// TIA Portal V17 export
// export: Created 2024-09-02T12:50:17.0977902Z, ExportSetting WithDefaults, DisplayName Totally Integrated Automation Portal, DisplayVersion V17, DisplayName TIA Portal Openness, DisplayVersion V17, DisplayName TIA Portal Version Control Interface, DisplayVersion V17, DisplayName STEP 7 Professional, DisplayVersion V17, DisplayName STEP 7 Safety, DisplayVersion V17, DisplayName WinCC Professional, DisplayVersion V17
DATA_BLOCK "AnwDB_ZP_InterfaceMainScreen_HMI1_OP70"   // DB160
{ S7_Optimized_Access := 'TRUE'; DB_Accessible_From_OPC_UA := 'FALSE' }
VERSION : 0.1
// stored: AutoNumber false, DBAccessibleFromOPCUA false, IsOnlyStoredInLoadMemory false, IsRetainMemResEnabled false, IsWriteProtectedInAS false, MemoryReserve 0
   VAR
      IsTactTime_Prestp : DInt;   // Isttaktzeit / Is tact time
      IsTactTime_Stp : DInt;   // Isttaktzeit / Is tact time
      Status : Struct   // Status Fremdgeraete / Status of external devices
         ExternalDevice_1 : Byte;   // Zustandsanzeige Fremdgerät 1 / Status display External device 1
         ExternalDevice_2 : Byte;   // Zustandsanzeige Fremdgerät 2 / Status display External device 2
         ExternalDevice_3 : Byte;   // Zustandsanzeige Fremdgerät 3 / Status display External device 3
         SLG_Station1 : Byte;   // Zustandsanzeige SLG an Station 1 / Status display SLG to Station 1
         SLG_Station2 : Byte;   // Zustandsanzeige SLG an Station 2 / Status display SLG to Station 2
         Reserve1 : Byte;
         Reserve2 : Byte;
         Reserve3 : Byte;
      END_STRUCT;
      Station : Array[0..1] of Struct   // Status Station / Status Station
         EStop : Bool;   // Anzeige Station Not Aus / Display station emergency stop
         Fault : Bool;   // Anzeige Station Störung / Display station fault
         SafetyDoor : Bool;   // Anzeige Station Schutztür / Display station Protective door
         TAF_deactivated : Bool;   // Anzeige Station TAF abgewählt / Display station TAF deselected
         Home : Bool;   // Anzeige Station Grundstellung / Station display Basic status
         Finished : Bool;   // Anzeige Station Fertig / Display Station Finished
      END_STRUCT;
      TransportRunning : Bool;   // Anzeige Transport läuft / Display Transport running
      Pallet_in_Station0 : Struct   // Werkstückträger am Vereinzeler / Workpiece carrier at separating stop
         Status : Int;   // Status
         TypeNr : Word := W#16#12;   // Typnummer / type number
         KeyNr : Word := W#16#4567;   // Schlüsselnummer / Button Number
         MotorNr : String[14] := 'ABC 1234567890';   // Motornummer / engine number
         WTNr : Word := W#16#8901;   // Werkstückträgernummer / workpiece carrier number
         RawPart : String[14] := 'XZY 1234567890';   // Rohteilbezeichnung / raw part designation
         PartPresent : Bool := true;   // Werkstückträger anwesend / Workpiece carrier present
         DataExist : Bool := true;   // Daten liegen vor / Data available
      END_STRUCT;
      Pallet_in_Station1 : Struct   // Werkstückträger in Station 1 / Workpiece carrier in station 1
         Status : Int := 4;   // Status
         TypeNr : Word := W#16#34;   // Typnummer / type number
         KeyNr : Word := W#16#8901;   // Schlüsselnummer / Button Number
         MotorNr : String[14] := 'ABC 1234567890';   // Motornummer / engine number
         WTNr : Word := W#16#2345;   // Werkstückträgernummer / workpiece carrier number
         RawPart : String[14] := 'XZY 1234567890';   // Rohteilbezeichnung / raw part designation
         PartPresent : Bool := true;   // Werkstückträger anwesend / Workpiece carrier present
         DataExist : Bool := true;   // Daten liegen vor / Data available
      END_STRUCT;
      Pallet_in_Station2 : Struct   // Werkstückträger in Station 2 / Workpiece carrier in station 2
         Status : Int;   // Status
         TypeNr : Word := W#16#56;   // Typnummer / type number
         KeyNr : Word := W#16#2345;   // Schlüsselnummer / Button Number
         MotorNr : String[14] := 'ABC 1234567890';   // Motornummer / engine number
         WTNr : Word := W#16#6789;   // Werkstückträgernummer / workpiece carrier number
         RawPart : String[14] := 'XZY 1234567890';   // Rohteilbezeichnung / raw part designation
         PartPresent : Bool := true;   // Werkstückträger anwesend / Workpiece carrier present
         DataExist : Bool := true;   // Daten liegen vor / Data available
      END_STRUCT;
      Pallet_in_Station3 : Struct   // Werkstückträger nach Station / Workpiece carrier by station
         Status : Int;   // Status
         TypeNr : Word := W#16#78;   // Typnummer / type number
         KeyNr : Word := W#16#6789;   // Schlüsselnummer / Button Number
         MotorNr : String[14] := 'ABC 1234567890';   // Motornummer / engine number
         WTNr : Word := W#16#123;   // Werkstückträgernummer / workpiece carrier number
         RawPart : String[14] := 'XZY 1234567890';   // Rohteilbezeichnung / raw part designation
         PartPresent : Bool := true;   // Werkstückträger anwesend / Workpiece carrier present
         DataExist : Bool := true;   // Daten liegen vor / Data available
      END_STRUCT;
      HMI_StatSummary { S7_SetPoint := 'True'} : "TypeSationsSum";   // Uebersicht MainScreen / Overview MainScreen
      HMI_PalletInfo { ExternalWritable := 'False'; S7_SetPoint := 'True'} : Array[1..8] of "TypeWTUebers_v2";   // Uebersicht WT Daten / Overview Pallet data
   END_VAR
BEGIN
   Station[0].EStop := TRUE;
   Station[0].Fault := TRUE;
   Station[0].SafetyDoor := TRUE;
   Station[0].TAF_deactivated := TRUE;
   Station[0].Home := TRUE;
   Station[0].Finished := TRUE;
END_DATA_BLOCK
